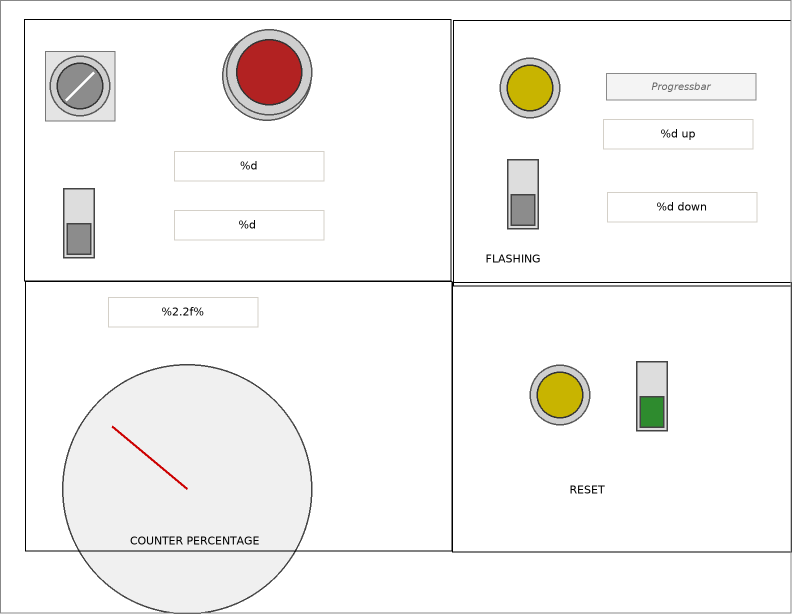
VISUALIZATION Visualization  // 792x614
    DipSwitch (44,188 70x70), variable: GVL.S1, behaviour: TOGGLE, style: Switch-DipSwitch-Gray
    RotarySwitch (45,51 70x70), variable: GVL.S2, behaviour: TOGGLE, style: Switch-RotarySwitch-Gray
    Lamp1 (215,23 104x106), variable: GVL.LED1, invisible if: GVL.S3, style: Lamp-Lamp1-Blue
    Textfield (174,151 150x30), "%d", text variable: GVL.counter
        OnDialogClosed: write the text variable via Default
    Textfield (174,210 150x30), "%d", text variable: MAIN1.counter1
        OnDialogClosed: write the text variable via Edit
    Lamp1 (495,53 70x70), variable: GVL.flasher, style: Lamp-Lamp1-Yellow
    DipSwitch (488,159 70x70), tooltip "%S", variable: GVL.S3, behaviour: TOGGLE, style: Switch-DipSwitch-Gray
    Textfield (603,119 150x30), "%d up", text variable: MAIN1.edge
    Textfield (607,192 150x30), "%d down", text variable: MAIN1.FALL
    DipSwitch (617,361 70x70), tooltip "reset", variable: GVL.S4, behaviour: TOGGLE, style: Switch-DipSwitch-Green
    Progressbar (606,73 150x27), variable: MAIN1.edge, invisible if: MAIN1.edge>50
    Lamp1 (215,22 108x100), variable: GVL.LED2, invisible if: GVL.LED1, style: Lamp-Lamp1-Red
    Lamp1 (525,360 70x70), variable: GVL.LED4, style: Lamp-Lamp1-Yellow
    Meter180 (62,364 250x250), value: GVL.counter/100, style: Meter-Meter180-Gray, scale format: %.1f, scale 0..100
    Label (120,509 150x64), "COUNTER PERCENTAGE"
    Label (512,475 150x30), "RESET"
    Label (438,244 150x30), "FLASHING"
    Rectangle (453,20 338x266)
    Rectangle (452,282 340x270)
    Rectangle (24,19 427x262)
    Rectangle (25,281 427x270)
    Textfield (108,297 150x30), "%2.2f%", text variable: GVL.counter/100.0
END_VISUALIZATION

(* stored: Version 1.1.0.1, ProductVersion 3.1.4024.12
   Visu Visualization: Id {dd173a1b-fe87-4c90-9ecd-275ff47a3dd1} *)
